INTERFACE I_AsyncRpcCallQueue

METHOD PUBLIC TryAddRpcCall : BOOL
VAR_INPUT
	CallingParameters : I_Deserializer;
	CallingAsynchronousRpcResponse : I_AsynchronousRpcResponse;
	CallingHandler : I_AsynchronousRpcHandler;
END_VAR
END_METHOD

END_INTERFACE

(* stored: Version 1.1.0.1, ProductVersion 3.1.4024.12
   Itf I_AsyncRpcCallQueue: Id {882bffff-5be5-4fb8-a5ce-d3269b93febb}
   Method TryAddRpcCall: Id {a7a4536c-a633-4dfa-b13e-c1da3d8f20a4} *)
